Staubli VAL3: MotionMode.pjx

--- MotionMode.pjx ---
Parameters version=s7.8.1 stackSize=5000 millimeterUnit=true
Program file=start.pgx
Program file=stop.pgx
Data file=MotionMode.dtx

--- MotionMode.dtx ---
public num JOINT_TRAJ
public num VELOCITY_CTRL
public num INVALID
